TYPE SimTimers_typ :
STRUCT
	// Orient
	TON_Orient_OpenBallClamp	: TON;
	TON_Orient_CloseBallClamp	: TON;
	TON_Orient_LoadBall			: TON;

	// Ball Seater
	TON_BallSeat_OpenBallClamp		: TON;
	TON_BallSeat_CloseBallClamp		: TON;
	TON_BallSeat_ExtendBallSeater	: TON;
	TON_BallSeat_RetractBallSeater	: TON;

	// Printer
	TON_Print_PrintComplete		: TON;
	
	// Vision
	TON_Vision_ScanBall		: TON;
	
	// Kickout
	TON_Kickout_OpenBallClamp		: TON;
	TON_Kickout_CloseBallClamp		: TON;
	TON_Kickout_RemoveBall			: TON;

	// Tray Load
	TON_TrayLoad_OpenBallClamp		: TON;
	TON_TrayLoad_CloseBallClamp		: TON;
	TON_TrayLoad_Complete			: TON;

END_STRUCT
END_TYPE

(* stored: Version 1.1.0.1, ProductVersion 3.1.4024.12
   DUT SimTimers_typ: Id {a900b90b-40d8-00c1-38f6-51cafb515166} *)
